// TIA Portal V19 export
TYPE "type_teachPara_plastic"
// stored: Access Published
   STRUCT
      U2Em2Cm5 : "type_teachPara_axis";
      U2Em4Cm1 { S7_SetPoint := 'True'} : "type_teachPara_axis";   // Xaxis
      U2Em4Cm2 { S7_SetPoint := 'True'} : "type_teachPara_axis";   // Yaxis
      U2Em4Cm3 { S7_SetPoint := 'True'} : "type_teachPara_axis";   // Zaxis
      U1Em2Cm5 : "type_teachPara_axis";
      U1Em4Cm1 { S7_SetPoint := 'True'} : "type_teachPara_axis";   // Xaxis
      U1Em4Cm2 { S7_SetPoint := 'True'} : "type_teachPara_axis";   // Yaxis
      U1Em4Cm3 { S7_SetPoint := 'True'} : "type_teachPara_axis";   // Zaxis
   END_STRUCT;
   // // U2Em2Cm5.position[0] : 24电芯 首位位置
   // // U2Em2Cm5.position[1] : 24电芯末尾位位置
   // // U2Em2Cm5.position[2] : 24 总长度 [1]-[0]
   // // U2Em2Cm5.position[3] : 36电芯 首位位置
   // // U2Em2Cm5.position[4] : 36电芯末尾位位置
   // // U2Em2Cm5.position[5] : 36 总长度 [1]-[0]
   // // U2Em2Cm5.position[20] : 24电芯 第一次顶位置
   // // U2Em2Cm5.position[21] : 24电芯 第二次顶位置
   // // U2Em2Cm5.position[22] : 24电芯 第三次顶位置
   // // U2Em2Cm5.position[30] : 36电芯 第1次顶位置
   // // U2Em2Cm5.position[31] : 36电芯 第2次顶位置
   // // U2Em2Cm5.position[32] : 36电芯 第3次顶位置
   // // U2Em2Cm5.position[33] : 36电芯 第4次顶位置
   // // U2Em2Cm5.position[34] : 36电芯 第5次顶位置
   // // U2Em4Cm1.position[0] : 24第一列电芯 首位位置
   // // U2Em4Cm1.position[1] : 24第一列电芯末尾位位置
   // // U2Em4Cm1.position[2] : 24 第1列总长度 [1]-[0]
   // // U2Em4Cm1.position[3] : 36第一列电芯 首位位置
   // // U2Em4Cm1.position[4] : 36第一列电芯末尾位位置
   // // U2Em4Cm1.position[5] : 36 第1列总长度 [1]-[0]
   // // U2Em4Cm1.position[6] : 24第2列电芯 首位位置
   // // U2Em4Cm1.position[7] : 24第2列电芯末尾位位置
   // // U2Em4Cm1.position[8] : 24 第2列总长度 [1]-[0]
   // // U2Em4Cm1.position[9] : 36第2列电芯 首位位置
   // // U2Em4Cm1.position[10] : 36第2列电芯末尾位位置
   // // U2Em4Cm1.position[11] : 36 第2列总长度 [1]-[0]
   // // U2Em4Cm1.position[12] : Xaxis
   // // U2Em4Cm1.position[13] : Xaxis
   // // U2Em4Cm1.position[14] : Xaxis
   // // U2Em4Cm1.position[15] : Xaxis
   // // U2Em4Cm1.position[16] : Xaxis
   // // U2Em4Cm1.position[17] : Xaxis
   // // U2Em4Cm1.position[18] : Xaxis
   // // U2Em4Cm1.position[19] : Xaxis
   // // U2Em4Cm1.position[20] : 24电芯 第一列电芯第一次顶位置
   // // U2Em4Cm1.position[21] : 24电芯 第一列电芯 第二次顶位置
   // // U2Em4Cm1.position[22] : 24电芯 第一列电芯第三次顶位置
   // // U2Em4Cm1.position[23] : Xaxis
   // // U2Em4Cm1.position[24] : Xaxis
   // // U2Em4Cm1.position[25] : Xaxis
   // // U2Em4Cm1.position[26] : Xaxis
   // // U2Em4Cm1.position[27] : Xaxis
   // // U2Em4Cm1.position[28] : Xaxis
   // // U2Em4Cm1.position[29] : Xaxis
   // // U2Em4Cm1.position[30] : 36电芯 第一列电芯第1次顶位置
   // // U2Em4Cm1.position[31] : 36电芯 第一列电芯第2次顶位置
   // // U2Em4Cm1.position[32] : 36电芯 第一列电芯第3次顶位置
   // // U2Em4Cm1.position[33] : 36电芯 第一列电芯第4次顶位置
   // // U2Em4Cm1.position[34] : 36电芯 第一列电芯第5次顶位置
   // // U2Em4Cm1.position[35] : Xaxis
   // // U2Em4Cm1.position[36] : Xaxis
   // // U2Em4Cm1.position[37] : Xaxis
   // // U2Em4Cm1.position[38] : Xaxis
   // // U2Em4Cm1.position[39] : Xaxis
   // // U2Em4Cm1.position[40] : 24电芯 第2列电芯第一次顶位置
   // // U2Em4Cm1.position[41] : 24电芯 第2列电芯 第二次顶位置
   // // U2Em4Cm1.position[42] : 24电芯 第2列电芯第三次顶位置
   // // U2Em4Cm1.position[43] : Xaxis
   // // U2Em4Cm1.position[44] : Xaxis
   // // U2Em4Cm1.position[45] : Xaxis
   // // U2Em4Cm1.position[46] : Xaxis
   // // U2Em4Cm1.position[47] : Xaxis
   // // U2Em4Cm1.position[48] : Xaxis
   // // U2Em4Cm1.position[49] : Xaxis
   // // U2Em4Cm1.position[50] : 36电芯 第2列电芯第1次顶位置
   // // U2Em4Cm1.position[51] : 36电芯 第2列电芯第2次顶位置
   // // U2Em4Cm1.position[52] : 36电芯 第2列电芯第3次顶位置
   // // U2Em4Cm1.position[53] : 36电芯 第2列电芯第4次顶位置
   // // U2Em4Cm1.position[54] : 36电芯 第2列电芯第5次顶位置
   // // U2Em4Cm2.position[0] : 24第一列电芯 首位位置
   // // U2Em4Cm2.position[1] : Yaxis
   // // U2Em4Cm2.position[2] : Yaxis
   // // U2Em4Cm2.position[3] : 36第一列电芯 首位位置
   // // U2Em4Cm2.position[4] : Yaxis
   // // U2Em4Cm2.position[5] : Yaxis
   // // U2Em4Cm2.position[6] : 24第2列电芯 首位位置
   // // U2Em4Cm2.position[7] : Yaxis
   // // U2Em4Cm2.position[8] : Yaxis
   // // U2Em4Cm2.position[9] : 36第2列电芯 首位位置
   // // U2Em4Cm3.position[0] : 下降位置
   // // U1Em2Cm5.position[0] : 24电芯 首位位置
   // // U1Em2Cm5.position[1] : 24电芯末尾位位置
   // // U1Em2Cm5.position[2] : 24 总长度 [1]-[0]
   // // U1Em2Cm5.position[3] : 36电芯 首位位置
   // // U1Em2Cm5.position[4] : 36电芯末尾位位置
   // // U1Em2Cm5.position[5] : 36 总长度 [1]-[0]
   // // U1Em2Cm5.position[20] : 24电芯 第一次顶位置
   // // U1Em2Cm5.position[21] : 24电芯 第二次顶位置
   // // U1Em2Cm5.position[22] : 24电芯 第三次顶位置
   // // U1Em2Cm5.position[30] : 36电芯 第1次顶位置
   // // U1Em2Cm5.position[31] : 36电芯 第2次顶位置
   // // U1Em2Cm5.position[32] : 36电芯 第3次顶位置
   // // U1Em2Cm5.position[33] : 36电芯 第4次顶位置
   // // U1Em2Cm5.position[34] : 36电芯 第5次顶位置
   // // U1Em4Cm1.position[0] : 24第一列电芯 首位位置
   // // U1Em4Cm1.position[1] : 24第一列电芯末尾位位置
   // // U1Em4Cm1.position[2] : 24 第1列总长度 [1]-[0]
   // // U1Em4Cm1.position[3] : 36第一列电芯 首位位置
   // // U1Em4Cm1.position[4] : 36第一列电芯末尾位位置
   // // U1Em4Cm1.position[5] : 36 第1列总长度 [1]-[0]
   // // U1Em4Cm1.position[6] : 24第2列电芯 首位位置
   // // U1Em4Cm1.position[7] : 24第2列电芯末尾位位置
   // // U1Em4Cm1.position[8] : 24 第2列总长度 [1]-[0]
   // // U1Em4Cm1.position[9] : 36第2列电芯 首位位置
   // // U1Em4Cm1.position[10] : 36第2列电芯末尾位位置
   // // U1Em4Cm1.position[11] : 36 第2列总长度 [1]-[0]
   // // U1Em4Cm1.position[12] : Xaxis
   // // U1Em4Cm1.position[13] : Xaxis
   // // U1Em4Cm1.position[14] : Xaxis
   // // U1Em4Cm1.position[15] : Xaxis
   // // U1Em4Cm1.position[16] : Xaxis
   // // U1Em4Cm1.position[17] : Xaxis
   // // U1Em4Cm1.position[18] : Xaxis
   // // U1Em4Cm1.position[19] : Xaxis
   // // U1Em4Cm1.position[20] : 24电芯 第一列电芯第一次顶位置
   // // U1Em4Cm1.position[21] : 24电芯 第一列电芯 第二次顶位置
   // // U1Em4Cm1.position[22] : 24电芯 第一列电芯第三次顶位置
   // // U1Em4Cm1.position[23] : Xaxis
   // // U1Em4Cm1.position[24] : Xaxis
   // // U1Em4Cm1.position[25] : Xaxis
   // // U1Em4Cm1.position[26] : Xaxis
   // // U1Em4Cm1.position[27] : Xaxis
   // // U1Em4Cm1.position[28] : Xaxis
   // // U1Em4Cm1.position[29] : Xaxis
   // // U1Em4Cm1.position[30] : 36电芯 第一列电芯第1次顶位置
   // // U1Em4Cm1.position[31] : 36电芯 第一列电芯第2次顶位置
   // // U1Em4Cm1.position[32] : 36电芯 第一列电芯第3次顶位置
   // // U1Em4Cm1.position[33] : 36电芯 第一列电芯第4次顶位置
   // // U1Em4Cm1.position[34] : 36电芯 第一列电芯第5次顶位置
   // // U1Em4Cm1.position[35] : Xaxis
   // // U1Em4Cm1.position[36] : Xaxis
   // // U1Em4Cm1.position[37] : Xaxis
   // // U1Em4Cm1.position[38] : Xaxis
   // // U1Em4Cm1.position[39] : Xaxis
   // // U1Em4Cm1.position[40] : 24电芯 第2列电芯第一次顶位置
   // // U1Em4Cm1.position[41] : 24电芯 第2列电芯 第二次顶位置
   // // U1Em4Cm1.position[42] : 24电芯 第2列电芯第三次顶位置
   // // U1Em4Cm1.position[43] : Xaxis
   // // U1Em4Cm1.position[44] : Xaxis
   // // U1Em4Cm1.position[45] : Xaxis
   // // U1Em4Cm1.position[46] : Xaxis
   // // U1Em4Cm1.position[47] : Xaxis
   // // U1Em4Cm1.position[48] : Xaxis
   // // U1Em4Cm1.position[49] : Xaxis
   // // U1Em4Cm1.position[50] : 36电芯 第2列电芯第1次顶位置
   // // U1Em4Cm1.position[51] : 36电芯 第2列电芯第2次顶位置
   // // U1Em4Cm1.position[52] : 36电芯 第2列电芯第3次顶位置
   // // U1Em4Cm1.position[53] : 36电芯 第2列电芯第4次顶位置
   // // U1Em4Cm1.position[54] : 36电芯 第2列电芯第5次顶位置
   // // U1Em4Cm2.position[0] : 24第一列电芯 首位位置
   // // U1Em4Cm2.position[1] : Yaxis
   // // U1Em4Cm2.position[2] : Yaxis
   // // U1Em4Cm2.position[3] : 36第一列电芯 首位位置
   // // U1Em4Cm2.position[4] : Yaxis
   // // U1Em4Cm2.position[5] : Yaxis
   // // U1Em4Cm2.position[6] : 24第2列电芯 首位位置
   // // U1Em4Cm2.position[7] : Yaxis
   // // U1Em4Cm2.position[8] : Yaxis
   // // U1Em4Cm2.position[9] : 36第2列电芯 首位位置
   // // U1Em4Cm3.position[0] : 下降位置
END_TYPE
